(* PLC project Generated.project, CODESYS CODESYS V3.5 SP19 Patch 1 *)
(* stored: creationDateTime 2026-08-30T22:32:01.336770, modificationDateTime 2026-08-30T22:32:01.336770 *)

(* ======================================================================= ST_fbDiveSearch_Inputs - Bus d'entree du cycle FB_DiveSearch ======================================================================= *)
TYPE ST_fbDiveSearch_Inputs : STRUCT
  PowerContactorEngaged : BOOL;  (* === AUTORISATIONS & COMMANDE === Chaine de puissance engagee *)
  Mode : E_Mode;  (* Mode arbitre courant *)
  MotionRequestActive : BOOL;  (* Demande de mouvement couplee *)
  MotionDirection : INT;  (* Sens demande (-1 = descente) *)
  BucketIsOpen : BOOL;  (* === CAPTEURS & MESURES === Benne ouverte confirmee *)
  KoboldImmersed : BOOL;  (* Kobold immerge *)
  M1Position_M : REAL;  (* Position cable M1 (m) *)
  M2Position_M : REAL;  (* Position cable M2 (m) *)
  PositionsValid : BOOL;  (* Mesures M1/M2 valides *)
  CurrentSpeedStep : INT;  (* Palier reel courant (0..5) *)
  DiveStartMin_M : REAL;  (* === REGLAGES METIER === Position minimale avant descente (m) *)
  ImmersionUpper_M : REAL;  (* Borne haute fenetre immersion (m) *)
  ImmersionLower_M : REAL;  (* Borne basse fenetre immersion (m) *)
  CableLimitAscent_M : REAL;  (* Limite haute exploitation (m) *)
  LimitLegalDepthMin_M : REAL;  (* Limite basse legale (m) *)
  CfgDiveFloorStep : INT;  (* Plancher palier descente (0..5) *)
  CycleTime : TIME;  (* Periode d'execution du cycle *)
  BypassPreconditions : BOOL;  (* Bypass reserve au mode maintenance N2/test *)
  Config : ST_fbDiveSearch_Config;  (* Parametres timeout *)
END_STRUCT;
END_TYPE

(* values of E_Mode: DISABLE: Mode Désactivé / Veille de sécurité (sorties bloquées); MAINT_N1: Manuel Niveau 1 : Pilotage unitaire avec toutes sécurités actives; MAINT_N2: Manuel Niveau 2 : Pilotage dégradé (droits étendus + bypasses autorisés); SEMI_AUTO: Mode Semi-Automatique (séquenceur automatique) *)

{attribute 'qualified_only'}
{attribute 'strict'}
TYPE E_Mode : (DISABLE := 0, MAINT_N1 := 1, MAINT_N2 := 2, SEMI_AUTO := 3);
END_TYPE

(* ======================================================================= ST_fbDiveSearch_Config - Reglages du cycle de recherche du fond ======================================================================= *)
TYPE ST_fbDiveSearch_Config : STRUCT
  DiveSpeedMin_Mps : REAL := 0.15;  (* Vitesse minimale de calcul du timeout (m/s) *)
  TimeoutMarginFactor : REAL := 1.5;  (* Marge appliquee au temps theorique *)
  TimeoutMinCourse_M : REAL := 1;  (* Course minimale prise en compte (m) *)
  TimeoutMaxCourse_M : REAL := 200;  (* Course maximale prise en compte (m) *)
  SecToMs : REAL := 1000;  (* Conversion secondes vers millisecondes *)
END_STRUCT;
END_TYPE
